(* CODESYS project GVL_POINT_MANAGER.gvl.xml

Project tree, tasks and I/O mapping:
  global variables GVL_POINT_MANAGER
*)

// GVL_POINT_MANAGER
{attribute 'qualified_only'}
VAR_GLOBAL
	PointManager : ST_POINT_MANAGER; // Команды, статусы и диагностика проверки точки
END_VAR
